// TIA Portal V20 export
// export: Created 2026-09-06T12:46:31.2345405Z, ExportSetting WithDefaults, DisplayName Totally Integrated Automation Portal, DisplayVersion V20, DisplayName TIA Portal Openness, DisplayVersion V20, DisplayName TIA Portal Version Control Interface, DisplayVersion V20, DisplayName STEP 7 Professional, DisplayVersion V20, DisplayName STEP 7 Safety, DisplayVersion V20, DisplayName WinCC Basic/Comfort/Advanced, DisplayVersion V20, DisplayName WinCC Professional, DisplayVersion V20, DisplayName WinCC Unified, DisplayVersion V20
DATA_BLOCK "Valve_Channels_DB"   // DB9
{ S7_Optimized_Access := 'TRUE' }
VERSION : 0.1
// Per-valve physical channel assignment, as six parallel flat arrays (one per UDT_Valve_Config field) rather than an array of the struct itself - Openness Import rejects StartValues on struct-typed array elements (confirmed via direct testing 2026-08-13, every encoding tried), while flat arrays of a simple type accept per-index StartValues cleanly, same as Valve_Meta_DB. Populated from the proposed station-by-zone channel assignment (AFT->ET200SP_AFT, ER->MID, FWD->FWD), reviewed and confirmed by the client before this import.
// stored: AutoNumber true, IsOnlyStoredInLoadMemory false, IsRetainMemResEnabled false, IsWriteProtectedInAS false, MemoryReserve 100
   VAR
      OpenFbChannel : Array[1..89] of Int;
      ClosedFbChannel : Array[1..89] of Int;
      HealthyChannel : Array[1..89] of Int;
      LocalModeChannel : Array[1..89] of Int;
      OpenCmdChannel : Array[1..89] of Int;
      CloseCmdChannel : Array[1..89] of Int;
   END_VAR
   VAR RETAIN
      TravelTimeout : Array[1..89] of Time;
      SeatBreakGrace : Array[1..89] of Time;
   END_VAR
BEGIN
   OpenFbChannel[1] := 1;
   OpenFbChannel[2] := 5;
   OpenFbChannel[3] := 9;
   OpenFbChannel[4] := 13;
   OpenFbChannel[5] := 17;
   OpenFbChannel[6] := 21;
   OpenFbChannel[7] := 25;
   OpenFbChannel[8] := 29;
   OpenFbChannel[9] := 33;
   OpenFbChannel[10] := 37;
   OpenFbChannel[11] := 41;
   OpenFbChannel[12] := 45;
   OpenFbChannel[13] := 49;
   OpenFbChannel[14] := 53;
   OpenFbChannel[15] := 57;
   OpenFbChannel[16] := 61;
   OpenFbChannel[17] := 65;
   OpenFbChannel[18] := 69;
   OpenFbChannel[19] := 73;
   OpenFbChannel[20] := 77;
   OpenFbChannel[21] := 81;
   OpenFbChannel[22] := 85;
   OpenFbChannel[23] := 89;
   OpenFbChannel[24] := 93;
   OpenFbChannel[25] := 97;
   OpenFbChannel[26] := 101;
   OpenFbChannel[27] := 105;
   OpenFbChannel[28] := 113;
   OpenFbChannel[29] := 117;
   OpenFbChannel[30] := 121;
   OpenFbChannel[31] := 125;
   OpenFbChannel[32] := 129;
   OpenFbChannel[33] := 133;
   OpenFbChannel[34] := 137;
   OpenFbChannel[35] := 141;
   OpenFbChannel[36] := 145;
   OpenFbChannel[37] := 149;
   OpenFbChannel[38] := 153;
   OpenFbChannel[39] := 157;
   OpenFbChannel[40] := 161;
   OpenFbChannel[41] := 165;
   OpenFbChannel[42] := 169;
   OpenFbChannel[43] := 173;
   OpenFbChannel[44] := 177;
   OpenFbChannel[45] := 181;
   OpenFbChannel[46] := 185;
   OpenFbChannel[47] := 189;
   OpenFbChannel[48] := 193;
   OpenFbChannel[49] := 197;
   OpenFbChannel[50] := 201;
   OpenFbChannel[51] := 205;
   OpenFbChannel[52] := 209;
   OpenFbChannel[53] := 213;
   OpenFbChannel[54] := 217;
   OpenFbChannel[55] := 225;
   OpenFbChannel[56] := 229;
   OpenFbChannel[57] := 233;
   OpenFbChannel[58] := 237;
   OpenFbChannel[59] := 241;
   OpenFbChannel[60] := 245;
   OpenFbChannel[61] := 249;
   OpenFbChannel[62] := 253;
   OpenFbChannel[63] := 257;
   OpenFbChannel[64] := 261;
   OpenFbChannel[65] := 265;
   OpenFbChannel[66] := 269;
   OpenFbChannel[67] := 273;
   OpenFbChannel[68] := 277;
   OpenFbChannel[69] := 281;
   OpenFbChannel[70] := 285;
   OpenFbChannel[71] := 289;
   OpenFbChannel[72] := 293;
   OpenFbChannel[73] := 297;
   OpenFbChannel[74] := 301;
   OpenFbChannel[75] := 305;
   OpenFbChannel[76] := 309;
   OpenFbChannel[77] := 313;
   OpenFbChannel[78] := 317;
   OpenFbChannel[79] := 321;
   OpenFbChannel[80] := 325;
   OpenFbChannel[81] := 329;
   OpenFbChannel[82] := 333;
   OpenFbChannel[83] := 337;
   OpenFbChannel[84] := 341;
   OpenFbChannel[85] := 345;
   OpenFbChannel[86] := 349;
   OpenFbChannel[87] := 353;
   OpenFbChannel[88] := 357;
   OpenFbChannel[89] := 361;
   ClosedFbChannel[1] := 2;
   ClosedFbChannel[2] := 6;
   ClosedFbChannel[3] := 10;
   ClosedFbChannel[4] := 14;
   ClosedFbChannel[5] := 18;
   ClosedFbChannel[6] := 22;
   ClosedFbChannel[7] := 26;
   ClosedFbChannel[8] := 30;
   ClosedFbChannel[9] := 34;
   ClosedFbChannel[10] := 38;
   ClosedFbChannel[11] := 42;
   ClosedFbChannel[12] := 46;
   ClosedFbChannel[13] := 50;
   ClosedFbChannel[14] := 54;
   ClosedFbChannel[15] := 58;
   ClosedFbChannel[16] := 62;
   ClosedFbChannel[17] := 66;
   ClosedFbChannel[18] := 70;
   ClosedFbChannel[19] := 74;
   ClosedFbChannel[20] := 78;
   ClosedFbChannel[21] := 82;
   ClosedFbChannel[22] := 86;
   ClosedFbChannel[23] := 90;
   ClosedFbChannel[24] := 94;
   ClosedFbChannel[25] := 98;
   ClosedFbChannel[26] := 102;
   ClosedFbChannel[27] := 106;
   ClosedFbChannel[28] := 114;
   ClosedFbChannel[29] := 118;
   ClosedFbChannel[30] := 122;
   ClosedFbChannel[31] := 126;
   ClosedFbChannel[32] := 130;
   ClosedFbChannel[33] := 134;
   ClosedFbChannel[34] := 138;
   ClosedFbChannel[35] := 142;
   ClosedFbChannel[36] := 146;
   ClosedFbChannel[37] := 150;
   ClosedFbChannel[38] := 154;
   ClosedFbChannel[39] := 158;
   ClosedFbChannel[40] := 162;
   ClosedFbChannel[41] := 166;
   ClosedFbChannel[42] := 170;
   ClosedFbChannel[43] := 174;
   ClosedFbChannel[44] := 178;
   ClosedFbChannel[45] := 182;
   ClosedFbChannel[46] := 186;
   ClosedFbChannel[47] := 190;
   ClosedFbChannel[48] := 194;
   ClosedFbChannel[49] := 198;
   ClosedFbChannel[50] := 202;
   ClosedFbChannel[51] := 206;
   ClosedFbChannel[52] := 210;
   ClosedFbChannel[53] := 214;
   ClosedFbChannel[54] := 218;
   ClosedFbChannel[55] := 226;
   ClosedFbChannel[56] := 230;
   ClosedFbChannel[57] := 234;
   ClosedFbChannel[58] := 238;
   ClosedFbChannel[59] := 242;
   ClosedFbChannel[60] := 246;
   ClosedFbChannel[61] := 250;
   ClosedFbChannel[62] := 254;
   ClosedFbChannel[63] := 258;
   ClosedFbChannel[64] := 262;
   ClosedFbChannel[65] := 266;
   ClosedFbChannel[66] := 270;
   ClosedFbChannel[67] := 274;
   ClosedFbChannel[68] := 278;
   ClosedFbChannel[69] := 282;
   ClosedFbChannel[70] := 286;
   ClosedFbChannel[71] := 290;
   ClosedFbChannel[72] := 294;
   ClosedFbChannel[73] := 298;
   ClosedFbChannel[74] := 302;
   ClosedFbChannel[75] := 306;
   ClosedFbChannel[76] := 310;
   ClosedFbChannel[77] := 314;
   ClosedFbChannel[78] := 318;
   ClosedFbChannel[79] := 322;
   ClosedFbChannel[80] := 326;
   ClosedFbChannel[81] := 330;
   ClosedFbChannel[82] := 334;
   ClosedFbChannel[83] := 338;
   ClosedFbChannel[84] := 342;
   ClosedFbChannel[85] := 346;
   ClosedFbChannel[86] := 350;
   ClosedFbChannel[87] := 354;
   ClosedFbChannel[88] := 358;
   ClosedFbChannel[89] := 362;
   HealthyChannel[1] := 3;
   HealthyChannel[2] := 7;
   HealthyChannel[3] := 11;
   HealthyChannel[4] := 15;
   HealthyChannel[5] := 19;
   HealthyChannel[6] := 23;
   HealthyChannel[7] := 27;
   HealthyChannel[8] := 31;
   HealthyChannel[9] := 35;
   HealthyChannel[10] := 39;
   HealthyChannel[11] := 43;
   HealthyChannel[12] := 47;
   HealthyChannel[13] := 51;
   HealthyChannel[14] := 55;
   HealthyChannel[15] := 59;
   HealthyChannel[16] := 63;
   HealthyChannel[17] := 67;
   HealthyChannel[18] := 71;
   HealthyChannel[19] := 75;
   HealthyChannel[20] := 79;
   HealthyChannel[21] := 83;
   HealthyChannel[22] := 87;
   HealthyChannel[23] := 91;
   HealthyChannel[24] := 95;
   HealthyChannel[25] := 99;
   HealthyChannel[26] := 103;
   HealthyChannel[27] := 107;
   HealthyChannel[28] := 115;
   HealthyChannel[29] := 119;
   HealthyChannel[30] := 123;
   HealthyChannel[31] := 127;
   HealthyChannel[32] := 131;
   HealthyChannel[33] := 135;
   HealthyChannel[34] := 139;
   HealthyChannel[35] := 143;
   HealthyChannel[36] := 147;
   HealthyChannel[37] := 151;
   HealthyChannel[38] := 155;
   HealthyChannel[39] := 159;
   HealthyChannel[40] := 163;
   HealthyChannel[41] := 167;
   HealthyChannel[42] := 171;
   HealthyChannel[43] := 175;
   HealthyChannel[44] := 179;
   HealthyChannel[45] := 183;
   HealthyChannel[46] := 187;
   HealthyChannel[47] := 191;
   HealthyChannel[48] := 195;
   HealthyChannel[49] := 199;
   HealthyChannel[50] := 203;
   HealthyChannel[51] := 207;
   HealthyChannel[52] := 211;
   HealthyChannel[53] := 215;
   HealthyChannel[54] := 219;
   HealthyChannel[55] := 227;
   HealthyChannel[56] := 231;
   HealthyChannel[57] := 235;
   HealthyChannel[58] := 239;
   HealthyChannel[59] := 243;
   HealthyChannel[60] := 247;
   HealthyChannel[61] := 251;
   HealthyChannel[62] := 255;
   HealthyChannel[63] := 259;
   HealthyChannel[64] := 263;
   HealthyChannel[65] := 267;
   HealthyChannel[66] := 271;
   HealthyChannel[67] := 275;
   HealthyChannel[68] := 279;
   HealthyChannel[69] := 283;
   HealthyChannel[70] := 287;
   HealthyChannel[71] := 291;
   HealthyChannel[72] := 295;
   HealthyChannel[73] := 299;
   HealthyChannel[74] := 303;
   HealthyChannel[75] := 307;
   HealthyChannel[76] := 311;
   HealthyChannel[77] := 315;
   HealthyChannel[78] := 319;
   HealthyChannel[79] := 323;
   HealthyChannel[80] := 327;
   HealthyChannel[81] := 331;
   HealthyChannel[82] := 335;
   HealthyChannel[83] := 339;
   HealthyChannel[84] := 343;
   HealthyChannel[85] := 347;
   HealthyChannel[86] := 351;
   HealthyChannel[87] := 355;
   HealthyChannel[88] := 359;
   HealthyChannel[89] := 363;
   LocalModeChannel[1] := 4;
   LocalModeChannel[2] := 8;
   LocalModeChannel[3] := 12;
   LocalModeChannel[4] := 16;
   LocalModeChannel[5] := 20;
   LocalModeChannel[6] := 24;
   LocalModeChannel[7] := 28;
   LocalModeChannel[8] := 32;
   LocalModeChannel[9] := 36;
   LocalModeChannel[10] := 40;
   LocalModeChannel[11] := 44;
   LocalModeChannel[12] := 48;
   LocalModeChannel[13] := 52;
   LocalModeChannel[14] := 56;
   LocalModeChannel[15] := 60;
   LocalModeChannel[16] := 64;
   LocalModeChannel[17] := 68;
   LocalModeChannel[18] := 72;
   LocalModeChannel[19] := 76;
   LocalModeChannel[20] := 80;
   LocalModeChannel[21] := 84;
   LocalModeChannel[22] := 88;
   LocalModeChannel[23] := 92;
   LocalModeChannel[24] := 96;
   LocalModeChannel[25] := 100;
   LocalModeChannel[26] := 104;
   LocalModeChannel[27] := 108;
   LocalModeChannel[28] := 116;
   LocalModeChannel[29] := 120;
   LocalModeChannel[30] := 124;
   LocalModeChannel[31] := 128;
   LocalModeChannel[32] := 132;
   LocalModeChannel[33] := 136;
   LocalModeChannel[34] := 140;
   LocalModeChannel[35] := 144;
   LocalModeChannel[36] := 148;
   LocalModeChannel[37] := 152;
   LocalModeChannel[38] := 156;
   LocalModeChannel[39] := 160;
   LocalModeChannel[40] := 164;
   LocalModeChannel[41] := 168;
   LocalModeChannel[42] := 172;
   LocalModeChannel[43] := 176;
   LocalModeChannel[44] := 180;
   LocalModeChannel[45] := 184;
   LocalModeChannel[46] := 188;
   LocalModeChannel[47] := 192;
   LocalModeChannel[48] := 196;
   LocalModeChannel[49] := 200;
   LocalModeChannel[50] := 204;
   LocalModeChannel[51] := 208;
   LocalModeChannel[52] := 212;
   LocalModeChannel[53] := 216;
   LocalModeChannel[54] := 220;
   LocalModeChannel[55] := 228;
   LocalModeChannel[56] := 232;
   LocalModeChannel[57] := 236;
   LocalModeChannel[58] := 240;
   LocalModeChannel[59] := 244;
   LocalModeChannel[60] := 248;
   LocalModeChannel[61] := 252;
   LocalModeChannel[62] := 256;
   LocalModeChannel[63] := 260;
   LocalModeChannel[64] := 264;
   LocalModeChannel[65] := 268;
   LocalModeChannel[66] := 272;
   LocalModeChannel[67] := 276;
   LocalModeChannel[68] := 280;
   LocalModeChannel[69] := 284;
   LocalModeChannel[70] := 288;
   LocalModeChannel[71] := 292;
   LocalModeChannel[72] := 296;
   LocalModeChannel[73] := 300;
   LocalModeChannel[74] := 304;
   LocalModeChannel[75] := 308;
   LocalModeChannel[76] := 312;
   LocalModeChannel[77] := 316;
   LocalModeChannel[78] := 320;
   LocalModeChannel[79] := 324;
   LocalModeChannel[80] := 328;
   LocalModeChannel[81] := 332;
   LocalModeChannel[82] := 336;
   LocalModeChannel[83] := 340;
   LocalModeChannel[84] := 344;
   LocalModeChannel[85] := 348;
   LocalModeChannel[86] := 352;
   LocalModeChannel[87] := 356;
   LocalModeChannel[88] := 360;
   LocalModeChannel[89] := 364;
   OpenCmdChannel[1] := 1;
   OpenCmdChannel[2] := 3;
   OpenCmdChannel[3] := 5;
   OpenCmdChannel[4] := 7;
   OpenCmdChannel[5] := 9;
   OpenCmdChannel[6] := 11;
   OpenCmdChannel[7] := 13;
   OpenCmdChannel[8] := 15;
   OpenCmdChannel[9] := 17;
   OpenCmdChannel[10] := 19;
   OpenCmdChannel[11] := 21;
   OpenCmdChannel[12] := 23;
   OpenCmdChannel[13] := 25;
   OpenCmdChannel[14] := 27;
   OpenCmdChannel[15] := 29;
   OpenCmdChannel[16] := 31;
   OpenCmdChannel[17] := 33;
   OpenCmdChannel[18] := 35;
   OpenCmdChannel[19] := 37;
   OpenCmdChannel[20] := 39;
   OpenCmdChannel[21] := 41;
   OpenCmdChannel[22] := 43;
   OpenCmdChannel[23] := 45;
   OpenCmdChannel[24] := 47;
   OpenCmdChannel[25] := 49;
   OpenCmdChannel[26] := 51;
   OpenCmdChannel[27] := 53;
   OpenCmdChannel[28] := 65;
   OpenCmdChannel[29] := 67;
   OpenCmdChannel[30] := 69;
   OpenCmdChannel[31] := 71;
   OpenCmdChannel[32] := 73;
   OpenCmdChannel[33] := 75;
   OpenCmdChannel[34] := 77;
   OpenCmdChannel[35] := 79;
   OpenCmdChannel[36] := 81;
   OpenCmdChannel[37] := 83;
   OpenCmdChannel[38] := 85;
   OpenCmdChannel[39] := 87;
   OpenCmdChannel[40] := 89;
   OpenCmdChannel[41] := 91;
   OpenCmdChannel[42] := 93;
   OpenCmdChannel[43] := 95;
   OpenCmdChannel[44] := 97;
   OpenCmdChannel[45] := 99;
   OpenCmdChannel[46] := 101;
   OpenCmdChannel[47] := 103;
   OpenCmdChannel[48] := 105;
   OpenCmdChannel[49] := 107;
   OpenCmdChannel[50] := 109;
   OpenCmdChannel[51] := 111;
   OpenCmdChannel[52] := 113;
   OpenCmdChannel[53] := 115;
   OpenCmdChannel[54] := 117;
   OpenCmdChannel[55] := 129;
   OpenCmdChannel[56] := 131;
   OpenCmdChannel[57] := 133;
   OpenCmdChannel[58] := 135;
   OpenCmdChannel[59] := 137;
   OpenCmdChannel[60] := 139;
   OpenCmdChannel[61] := 141;
   OpenCmdChannel[62] := 143;
   OpenCmdChannel[63] := 145;
   OpenCmdChannel[64] := 147;
   OpenCmdChannel[65] := 149;
   OpenCmdChannel[66] := 151;
   OpenCmdChannel[67] := 153;
   OpenCmdChannel[68] := 155;
   OpenCmdChannel[69] := 157;
   OpenCmdChannel[70] := 159;
   OpenCmdChannel[71] := 161;
   OpenCmdChannel[72] := 163;
   OpenCmdChannel[73] := 165;
   OpenCmdChannel[74] := 167;
   OpenCmdChannel[75] := 169;
   OpenCmdChannel[76] := 171;
   OpenCmdChannel[77] := 173;
   OpenCmdChannel[78] := 175;
   OpenCmdChannel[79] := 177;
   OpenCmdChannel[80] := 179;
   OpenCmdChannel[81] := 181;
   OpenCmdChannel[82] := 183;
   OpenCmdChannel[83] := 185;
   OpenCmdChannel[84] := 187;
   OpenCmdChannel[85] := 189;
   OpenCmdChannel[86] := 191;
   OpenCmdChannel[87] := 193;
   OpenCmdChannel[88] := 195;
   OpenCmdChannel[89] := 197;
   CloseCmdChannel[1] := 2;
   CloseCmdChannel[2] := 4;
   CloseCmdChannel[3] := 6;
   CloseCmdChannel[4] := 8;
   CloseCmdChannel[5] := 10;
   CloseCmdChannel[6] := 12;
   CloseCmdChannel[7] := 14;
   CloseCmdChannel[8] := 16;
   CloseCmdChannel[9] := 18;
   CloseCmdChannel[10] := 20;
   CloseCmdChannel[11] := 22;
   CloseCmdChannel[12] := 24;
   CloseCmdChannel[13] := 26;
   CloseCmdChannel[14] := 28;
   CloseCmdChannel[15] := 30;
   CloseCmdChannel[16] := 32;
   CloseCmdChannel[17] := 34;
   CloseCmdChannel[18] := 36;
   CloseCmdChannel[19] := 38;
   CloseCmdChannel[20] := 40;
   CloseCmdChannel[21] := 42;
   CloseCmdChannel[22] := 44;
   CloseCmdChannel[23] := 46;
   CloseCmdChannel[24] := 48;
   CloseCmdChannel[25] := 50;
   CloseCmdChannel[26] := 52;
   CloseCmdChannel[27] := 54;
   CloseCmdChannel[28] := 66;
   CloseCmdChannel[29] := 68;
   CloseCmdChannel[30] := 70;
   CloseCmdChannel[31] := 72;
   CloseCmdChannel[32] := 74;
   CloseCmdChannel[33] := 76;
   CloseCmdChannel[34] := 78;
   CloseCmdChannel[35] := 80;
   CloseCmdChannel[36] := 82;
   CloseCmdChannel[37] := 84;
   CloseCmdChannel[38] := 86;
   CloseCmdChannel[39] := 88;
   CloseCmdChannel[40] := 90;
   CloseCmdChannel[41] := 92;
   CloseCmdChannel[42] := 94;
   CloseCmdChannel[43] := 96;
   CloseCmdChannel[44] := 98;
   CloseCmdChannel[45] := 100;
   CloseCmdChannel[46] := 102;
   CloseCmdChannel[47] := 104;
   CloseCmdChannel[48] := 106;
   CloseCmdChannel[49] := 108;
   CloseCmdChannel[50] := 110;
   CloseCmdChannel[51] := 112;
   CloseCmdChannel[52] := 114;
   CloseCmdChannel[53] := 116;
   CloseCmdChannel[54] := 118;
   CloseCmdChannel[55] := 130;
   CloseCmdChannel[56] := 132;
   CloseCmdChannel[57] := 134;
   CloseCmdChannel[58] := 136;
   CloseCmdChannel[59] := 138;
   CloseCmdChannel[60] := 140;
   CloseCmdChannel[61] := 142;
   CloseCmdChannel[62] := 144;
   CloseCmdChannel[63] := 146;
   CloseCmdChannel[64] := 148;
   CloseCmdChannel[65] := 150;
   CloseCmdChannel[66] := 152;
   CloseCmdChannel[67] := 154;
   CloseCmdChannel[68] := 156;
   CloseCmdChannel[69] := 158;
   CloseCmdChannel[70] := 160;
   CloseCmdChannel[71] := 162;
   CloseCmdChannel[72] := 164;
   CloseCmdChannel[73] := 166;
   CloseCmdChannel[74] := 168;
   CloseCmdChannel[75] := 170;
   CloseCmdChannel[76] := 172;
   CloseCmdChannel[77] := 174;
   CloseCmdChannel[78] := 176;
   CloseCmdChannel[79] := 178;
   CloseCmdChannel[80] := 180;
   CloseCmdChannel[81] := 182;
   CloseCmdChannel[82] := 184;
   CloseCmdChannel[83] := 186;
   CloseCmdChannel[84] := 188;
   CloseCmdChannel[85] := 190;
   CloseCmdChannel[86] := 192;
   CloseCmdChannel[87] := 194;
   CloseCmdChannel[88] := 196;
   CloseCmdChannel[89] := 198;
   TravelTimeout[1..89] := T#60s;
   SeatBreakGrace[1..89] := T#10s;
END_DATA_BLOCK
